FUNCTION_BLOCK FB_Normalize
VAR_INPUT
	nRawInput : INT;
	fMaxValue : LREAL;
END_VAR
VAR_OUTPUT
	fNormalizedInput : LREAL;
END_VAR
VAR
END_VAR

fNormalizedInput := (fMaxValue	* INT_TO_LREAL(nRawInput)) / 32767.0;

fNormalizedInput := LIMIT(0, fNormalizedInput, fMaxValue);

END_FUNCTION_BLOCK

(* stored: Version 1.1.0.1, ProductVersion 3.1.4024.13
   POU FB_Normalize: Id {72f82d73-0f72-40ed-bb1d-a8162c2cf4db}, SpecialFunc None *)
